{attribute 'linkalways'}
{attribute 'hide_all_locals'}
FUNCTION_BLOCK ValueUdintRead EXTENDS ValueBase IMPLEMENTS ValueRead
VAR
	thisValue : UDINT;
END_VAR

{attribute 'call_after_global_init_slot' := '1'}
{attribute 'call_after_online_change_slot' := '1'}
METHOD PROTECTED GetThisAnyType
VAR_INPUT
END_VAR
thisAnyType := ToAnyType(thisValue);
END_METHOD

METHOD GetAsType : BOOL
VAR_INPUT
	destination : __SYSTEM.AnyType;
END_VAR
GetAsType := ConvertAnyType(thisAnyType, destination);
END_METHOD

METHOD GetAsString : T_MaxString
VAR_INPUT
END_VAR
GetAsString := TO_STRING(thisValue);
END_METHOD

METHOD Get : BOOL
VAR_INPUT
	destination : ANY;
END_VAR
Get := ConvertAnyType(thisAnyType, destination);
END_METHOD

METHOD FB_init : BOOL
VAR_INPUT
	bInitRetains : BOOL; // if TRUE, the retain variables are initialized (warm start / cold start)
	bInCopyCode : BOOL;  // if TRUE, the instance afterwards gets moved into the copy code (online change)
END_VAR
_ValueType := __SYSTEM.TYPE_CLASS.TYPE_UDINT;
END_METHOD

{attribute 'monitoring' := 'call'}
PROPERTY Value : UDINT
GET
Value := thisValue;
END_GET
END_PROPERTY

END_FUNCTION_BLOCK

(* stored: Version 1.1.0.1
   POU ValueUdintRead: Id {741b6723-5ddd-436e-8099-f9b932ff423a}, SpecialFunc None
   Method GetThisAnyType: Id {a36445ee-6984-4d47-ad4d-89d34ad9b645}
   Method GetAsType: Id {83198f2c-9aa7-40a8-b4b1-706c06555234}
   Method GetAsString: Id {03b77400-09bb-4e10-a549-c162ba04e42b}
   Method Get: Id {75e3fe00-898a-42ba-bfdb-0bcfba065564}
   Method FB_init: Id {726a7557-82f0-460d-b974-80df13a4c44e}
   Property Value: Id {1a86ec39-f675-4d46-a7d3-7141d1b66ade}
   Get Get: Id {e65eb884-9988-4580-b8db-f3dea34365d0} *)
